// TIA Portal V19 export
VAR_GLOBAL   // PLC tag table "DemoCaseTags"
   POT4_G120 AT %MD30 : Real;
   HMI_IO_Test AT %M10.4 : Bool;
   PB_Green_1200 AT %M60.0 : Bool;
   PB_Blue_1200 AT %M60.1 : Bool;
   POT3_Upper_1200 AT %MW62 : Int;
   PB_Green_Lamp_1200 AT %M64.0 : Bool;
   PB_Blue_Lamp_1200 AT %M64.1 : Bool;
   TopLights_Green_1200 AT %M64.5 : Bool;
   TopLights_Red_1200 AT %M64.6 : Bool;
   TopLights_Blue_1200 AT %M64.7 : Bool;
   "1200_Inputs" AT %MB60 : Byte;
   "1200_Outputs" AT %MB64 : Byte;
   "1200_All_Inputs" AT %MD60 : DWord;
   OS6 AT %M11.4 : Bool;
   "Red Latch" AT %M11.5 : Bool;
   "Green Latch" AT %M11.6 : Bool;
   GateClosed AT %M11.7 : Bool;
   "Blue Latch" AT %M20.3 : Bool;
   Coordination AT %MW36 : Int;
   POT2_Warning AT %M20.4 : Bool;
END_VAR
